# EPICS SNL sequencer program: mpgSupport/src/edefMask.st
program edefMask

option -a;  /* All pvGets must be synchronous */
option +c;  /* All connections must be made before execution begins */
option +d;  /* Turn on runtime debug messages */

%%#include <string.h> 	   /* sprintf prototype */

int maskChanged;
assign maskChanged to "{IOC}:MASKCHG";
monitor maskChanged;
evflag maskChanged_ef;
sync maskChanged maskChanged_ef;

int bitChanged;
assign bitChanged to "{IOC}:BITCHG";
monitor bitChanged;
evflag bitChanged_ef;
sync bitChanged bitChanged_ef;

unsigned long dgrpINCM[3];
assign dgrpINCM to "VX00:DGRP:1150:INCM";
monitor dgrpINCM;

unsigned long dgrpEXCM[3];
assign dgrpEXCM to "VX00:DGRP:1150:EXCM";
monitor dgrpEXCM;

int initDone;
assign initDone to "{IOC}:MASKSETUP";

unsigned short dgrpSHORT;
short i;
short j;
short eachBit;
short bitp;
short savedINCM[20][160];
short savedEXCM[20][160];

int edefMaxNumber;
int edefNumber;

int maskMaxNumber;
int maskCount;
int maskNumber;
int maskVal;

int pnbnMaxNumber;
int pnbnNumber;

string NAMEval;
assign NAMEval to "";
string NAMEpv;

string PNBNval;
assign PNBNval to "";
string PNBNpv;

int BITPval;
assign BITPval to "";
string BITPpv;

int BITWval;
assign BITWval to "";
string BITWpv;

string DESCval;
assign DESCval to "";
string DESCpv;

string DESC1val;
assign DESC1val to "";
string DESC1pv;

int INCMval;
assign INCMval to "";
string INCMpv;

int EXCMval;
assign EXCMval to "";
string EXCMpv;

string INCMSval;
assign INCMSval to "";
string INCMSpv;
int iINCMS;

string EXCMSval;
assign EXCMSval to "";
string EXCMSpv;
int iEXCMS;

unsigned long INCLUSIONval;
assign INCLUSIONval to "";
string INCLUSIONpv;

unsigned long EXCLUSIONval;
assign EXCLUSIONval to "";
string EXCLUSIONpv;

unsigned short INCLUSIONvalSHORT;
assign INCLUSIONvalSHORT to "";
string INCLUSIONpvSHORT;

unsigned short EXCLUSIONvalSHORT;
assign EXCLUSIONvalSHORT to "";
string EXCLUSIONpvSHORT;

int sort_done;
int debug_flag;

char * SYS;

entry {

  debug_flag = 0;
  if (debug_flag) printf ("edefMask:entry\n");

  sort_done = 0;

  edefMaxNumber = 20;
  edefNumber = 0;

  maskMaxNumber = 160;
  maskCount = 0;
  maskNumber = 0;

  pnbnMaxNumber = 124;
  pnbnNumber = 0;
  sprintf (PNBNval, "");

  SYS = macValueGet("SYS");

  } /* edefMask entry*/

ss edefMaskStateSet {

  state pnbn_read {

    entry {
      if (debug_flag) printf ("edefMaskStateSet:pnbn_read");

      /* setup first PNBN NAME, BITP & BITW */
      pnbnNumber++;
      sprintf (PNBNpv, "MP00:PNBN:%d:NAME", pnbnNumber);
      pvAssign (PNBNval, PNBNpv);
      pvMonitor (PNBNval);

      BITPval = -1;
      sprintf (BITPpv, "MP00:PNBN:%d:BITP", pnbnNumber);
      pvAssign (BITPval, BITPpv);
      pvMonitor (BITPval);

      BITWval = -1;
      sprintf (BITWpv, "MP00:PNBN:%d:BITW", pnbnNumber);
      pvAssign (BITWval, BITWpv);
      pvMonitor (BITWval);
      } /* pnbn_read entry */

    when (pnbnNumber > pnbnMaxNumber) {
      } state pnbn_sort

    when ((strlen(PNBNval)>0) && (BITPval>-1) && (BITWval>-1)) {
      if ((BITPval < 32) || (0 == strncmp ("            ", PNBNval, 12))) {
        /* unused PNBN name, 32 comes from PNET_MODFBIT_LOLIM */
        }
      else {
        if (debug_flag) printf (".");
        maskCount++;
        /* Put the name in INCM DESC */
        sprintf (DESC1pv, "EDEF:%s:1:INCM%d.DESC", SYS, maskCount);
        pvAssign (DESC1val, DESC1pv);
        sprintf (DESC1val, "%s", PNBNval);
        pvPut (DESC1val);
        /* Put the BITP & BITW into the EXCM DESC */
        sprintf (DESC1pv, "EDEF:%s:1:EXCM%d.DESC", SYS, maskCount);
        pvAssign (DESC1val, DESC1pv);
        sprintf (DESC1val, "%3.3d %3.3d", BITPval, BITWval);
        pvPut (DESC1val);
        }; /* non-blank pnbn name */
      pnbnNumber++;
      sprintf (PNBNval, "");
      BITPval = -1;
      BITWval = -1;
      if (pnbnNumber <= pnbnMaxNumber) {
        sprintf (PNBNpv, "MP00:PNBN:%d:NAME", pnbnNumber);
        pvAssign (PNBNval, PNBNpv);
        pvMonitor (PNBNval);
        sprintf (BITPpv, "MP00:PNBN:%d:BITP", pnbnNumber);
        pvAssign (BITPval, BITPpv);
        pvMonitor (BITPval);
        sprintf (BITWpv, "MP00:PNBN:%d:BITW", pnbnNumber);
        pvAssign (BITWval, BITWpv);
        pvMonitor (BITWval);
        }; /* setup next pnbn unit */
      } state pnbn_read
    } /* state pnbn_read */

  state pnbn_sort {
    entry {
      if (debug_flag) printf ("\nedefMaskStateSet:pnbn_sort");
      }
    when (sort_done) {
      } state pnbn_assign
    when (1) {
      if (debug_flag) printf (".");
      sort_done = 1;
      for (maskNumber = 1; maskNumber < maskCount; maskNumber++) {
        sprintf (DESC1pv, "EDEF:%s:1:INCM%d.DESC", SYS, maskNumber);
        pvAssign (DESC1val, DESC1pv);
        pvGet (DESC1val);
        sprintf (DESCpv, "EDEF:%s:1:INCM%d.DESC", SYS, 1+maskNumber);
        pvAssign (DESCval, DESCpv);
        pvGet (DESCval);
        if (strcmp (DESC1val, DESCval) > 0) {
          sort_done = 0;
          /* switch INCM DESC's */
          sprintf (PNBNval, "%s", DESC1val);
          sprintf (DESC1val, "%s", DESCval);
          sprintf (DESCval, "%s", PNBNval);
          pvPut (DESC1val);
          pvPut (DESCval);
          /* switch EXCM DESC's */
          sprintf (DESC1pv, "EDEF:%s:1:EXCM%d.DESC", SYS, maskNumber);
          pvAssign (DESC1val, DESC1pv);
          pvGet (DESC1val);
          sprintf (DESCpv, "EDEF:%s:1:EXCM%d.DESC", SYS, 1+maskNumber);
          pvAssign (DESCval, DESCpv);
          pvGet (DESCval);
          sprintf (PNBNval, "%s", DESC1val);
          sprintf (DESC1val, "%s", DESCval);
          sprintf (DESCval, "%s", PNBNval);
          pvPut (DESC1val);
          pvPut (DESCval);
          }; /* switch */
        }; /* for each mask */
      } state pnbn_sort
    } /* state pnbn sort */

  state pnbn_assign {
    entry {
      if (debug_flag) printf ("\nedefMaskStateSet:pnbn_assign\n");
      }
    when (1) {
      for (maskNumber = 1; maskNumber <= maskCount; maskNumber++) {
        sprintf (DESC1pv, "EDEF:%s:1:INCM%d.DESC", SYS, maskNumber);
        pvAssign (DESC1val, DESC1pv);
        pvGet (DESC1val);
        for (edefNumber = 2; edefNumber <= edefMaxNumber; edefNumber++) {
          sprintf (DESCpv, "EDEF:%s:%d:INCM%d.DESC", SYS, edefNumber, maskNumber);
          pvAssign (DESCval, DESCpv);
          sprintf (DESCval, "%s", DESC1val);
          pvPut (DESCval);
          }; /* for each edef */
        }; /* for each mask */
      for (maskNumber = 1; maskNumber <= maskCount; maskNumber++) {
        sprintf (DESC1pv, "EDEF:%s:1:EXCM%d.DESC", SYS, maskNumber);
        pvAssign (DESC1val, DESC1pv);
        pvGet (DESC1val);
        for (edefNumber = 2; edefNumber <= edefMaxNumber; edefNumber++) {
          sprintf (DESCpv, "EDEF:%s:%d:EXCM%d.DESC", SYS, edefNumber, maskNumber);
          pvAssign (DESCval, DESCpv);
          sprintf (DESCval, "%s", DESC1val);
          pvPut (DESCval);
          }; /* for each edef */
        }; /* for each mask */
      } state dgrp_incm_excm_set
    } /* state pnbn assign */

  state dgrp_incm_excm_set {
    entry {
      if (debug_flag) printf ("edefMaskStateSet:dgrp_incm_excm_set\n");
      }
    /* read DGRP INCM & EXCM and set INCLUSION[1..5][A|B] & EXCLUSION[1..5][A|B] */
    when (1) {
      for (i=0; i<3; i++) {
        for (edefNumber = 1; edefNumber <= edefMaxNumber; edefNumber++) {
          dgrpSHORT = dgrpINCM[i] & 0x0000FFFF;
          sprintf (INCLUSIONpvSHORT, "EDEF:%s:%d:INCLUSION%dA", SYS, edefNumber, 1+i);
          pvAssign (INCLUSIONvalSHORT, INCLUSIONpvSHORT);
          INCLUSIONvalSHORT = dgrpSHORT;
          pvPut (INCLUSIONvalSHORT);

          dgrpSHORT = (dgrpINCM[i] & 0xFFFF0000) >> 16;
          sprintf (INCLUSIONpvSHORT, "EDEF:%s:%d:INCLUSION%dB", SYS, edefNumber, 1+i);
          pvAssign (INCLUSIONvalSHORT, INCLUSIONpvSHORT);
          INCLUSIONvalSHORT = dgrpSHORT;
          pvPut (INCLUSIONvalSHORT);

          dgrpSHORT = dgrpEXCM[i] & 0x0000FFFF;
          sprintf (EXCLUSIONpvSHORT, "EDEF:%s:%d:EXCLUSION%dA", SYS, edefNumber, 1+i);
          pvAssign (EXCLUSIONvalSHORT, EXCLUSIONpvSHORT);
          EXCLUSIONvalSHORT = dgrpSHORT;
          pvPut (EXCLUSIONvalSHORT);

          dgrpSHORT = (dgrpEXCM[i] & 0xFFFF0000) >> 16;
          sprintf (EXCLUSIONpvSHORT, "EDEF:%s:%d:EXCLUSION%dB", SYS, edefNumber, 1+i);
          pvAssign (EXCLUSIONvalSHORT, EXCLUSIONpvSHORT);
          EXCLUSIONvalSHORT = dgrpSHORT;
          pvPut (EXCLUSIONvalSHORT);
          }; /* for each edef */
        };
        sprintf (INCMSval, "1HZ");
        sprintf (PNBNval, "ONE_HERTZ");
      } state special_incm_excm_set
    } /* state dgrp_incm_excm_set */

  state special_incm_excm_set {
    /* Look for 1Hz and 10Hz eDefs and set their ONE_HERTZ & TEN_HERTZ INCLUSION[1..5][A|B] */
    entry {
      if (debug_flag) printf ("edefMaskStateSet:special_incm_excm_set\n");
      }
    when (0 == strlen(INCMSval)) {
      } state incm_excm_set
    when (1) {
      for (edefNumber = 1; edefNumber <= edefMaxNumber; edefNumber++) {
        sprintf (NAMEpv, "EDEF:%s:%d:NAME", SYS, edefNumber);
        pvAssign (NAMEval, NAMEpv);
        pvGet (NAMEval);
        if (0 == strncmp (NAMEval, INCMSval, strlen(INCMSval))) {
          for (maskNumber = 1; maskNumber <= maskCount; maskNumber++) {
            sprintf (DESCpv, "EDEF:%s:%d:INCM%d.DESC", SYS, edefNumber, maskNumber);
            pvAssign (DESCval, DESCpv);
            pvGet (DESCval);
            if (0 == strncmp (DESCval, PNBNval, strlen(PNBNval))) {
              sprintf (DESCpv, "EDEF:%s:%d:EXCM%d.DESC", SYS, edefNumber, maskNumber);
              pvAssign (DESCval, DESCpv);
              pvGet (DESCval);
              sscanf (DESCval, "%3d %3d", &BITPval, &BITWval);
              for (eachBit = 0; eachBit < BITWval; eachBit++) {
                bitp = BITPval + eachBit;
                j = 0; /* EDEF:SYS:[edefNumbner]:INCLUSION[j] */
                while (bitp > 31) {
                  j++;
                  bitp = bitp - 32;
                  };
                if (bitp < 16) {
                  sprintf (INCLUSIONpvSHORT, "EDEF:%s:%d:INCLUSION%dA", SYS, edefNumber, j);
                  pvAssign (INCLUSIONvalSHORT, INCLUSIONpvSHORT);
                  pvGet (INCLUSIONvalSHORT);
                  INCLUSIONvalSHORT += (1 << bitp);
                  pvPut (INCLUSIONvalSHORT);
                  }
                else {
                  sprintf (INCLUSIONpvSHORT, "EDEF:%s:%d:INCLUSION%dB", SYS, edefNumber, j);
                  pvAssign (INCLUSIONvalSHORT, INCLUSIONpvSHORT);
                  pvGet (INCLUSIONvalSHORT);
                  bitp = bitp - 16;
                  INCLUSIONvalSHORT += (1 << bitp);
                  pvPut (INCLUSIONvalSHORT);
                  };
                }; /* for each BITW */
              }; /* Found mask name */
            }; /* each mask */
          }; /* found correct EDEF NAME */
        }; /* each edef */
      if (0 == strcmp (INCMSval, "1HZ")) {
        sprintf (INCMSval, "10HZ");
        sprintf (PNBNval, "TEN_HERTZ");
        }
      else {
        sprintf (INCMSval, "");
        initDone = 1;
        pvPut (initDone);
        };
      } state special_incm_excm_set
    } /* state special_incm_excm */

  state incm_excm_set {
    /* Set INCMS[1..4] & EXCMS[1..4] and INCM[1..maskCount] & EXCM[1..maskCount]
       based on INCLUSION[1..5] EXCLUSION[1..5] */
    entry {
      if (debug_flag) printf ("edefMaskStateSet:incm_excm_set\n");
      }
    when(1) {
      for (edefNumber = 1; edefNumber <= edefMaxNumber; edefNumber++) {
        iINCMS=1;
        sprintf (INCMSpv, "EDEF:%s:%d:INCMS%d", SYS, edefNumber, iINCMS);
        pvAssign (INCMSval, INCMSpv);
        sprintf (INCMSval, "");
        iEXCMS=1;
        sprintf (EXCMSpv, "EDEF:%s:%d:EXCMS%d", SYS, edefNumber, iEXCMS);
        pvAssign (EXCMSval, EXCMSpv);
        sprintf (EXCMSval, "");
        for (maskNumber = 1; maskNumber <= maskCount; maskNumber++) {
          i = 0; /* index into INCLUSION & EXCLUSION */
          /* Is my BITP set? */
          sprintf (DESCpv, "EDEF:%s:%d:EXCM%d.DESC", SYS, edefNumber, maskNumber);
          pvAssign (DESCval, DESCpv);
          pvGet (DESCval);
          sscanf (DESCval, "%3d", &BITPval);
          sprintf (DESCpv, "EDEF:%s:%d:INCM%d.DESC", SYS, edefNumber, maskNumber);
          pvAssign (DESCval, DESCpv);
          pvGet (DESCval);
          sprintf (PNBNval, "%s", DESCval); /* remove trailing blanks */
          for (j=0; j<sizeof(PNBNval); j++) if (' ' == PNBNval[j]) PNBNval[j]=0;
          pvGet (DESCval);
          while (BITPval > 31) {
            i++;
            BITPval = BITPval - 32;
            };
          sprintf (INCLUSIONpv, "EDEF:%s:%d:INCLUSION%d", SYS, edefNumber, i);
          pvAssign (INCLUSIONval, INCLUSIONpv);
          pvGet (INCLUSIONval);
          sprintf (EXCLUSIONpv, "EDEF:%s:%d:EXCLUSION%d", SYS, edefNumber, i);
          pvAssign (EXCLUSIONval, EXCLUSIONpv);
          pvGet (EXCLUSIONval);
          sprintf (INCMpv, "EDEF:%s:%d:INCM%d", SYS, edefNumber, maskNumber);
          pvAssign (INCMval, INCMpv);
          pvGet (INCMval);
          sprintf (EXCMpv, "EDEF:%s:%d:EXCM%d", SYS, edefNumber, maskNumber);
          pvAssign (EXCMval, EXCMpv);
          pvGet (EXCMval);
          if (INCLUSIONval & (1 << BITPval)) {
            maskVal = 1;
            if ((strlen(INCMSval) + strlen(PNBNval)) > 38) {
              pvPut (INCMSval);
              sprintf (INCMSpv, "EDEF:%s:%d:INCMS%d", SYS, edefNumber, ++iINCMS);
              pvAssign (INCMSval, INCMSpv);
              sprintf (INCMSval, "");
              };
            if (iINCMS < 5) {
              if (0 == strlen(INCMSval)) {
                sprintf (INCMSval, "%s", PNBNval);
                }
              else {
                strcat (INCMSval, " ");
                strcat (INCMSval, PNBNval);
                };
              };
            } /* INCLUSION bit set */
          else {
            maskVal = 0;
            }; /* INCLUSION bit not set */
          if (maskVal != INCMval) {
            INCMval = maskVal;
            pvPut(INCMval);
            };
          if (EXCLUSIONval & (1 << BITPval)) {
            maskVal = 1;
            if ((strlen(EXCMSval) + strlen(PNBNval)) > 38) {
              pvPut (EXCMSval);
              sprintf (EXCMSpv, "EDEF:%s:%d:EXCMS%d", SYS, edefNumber, ++iEXCMS);
              pvAssign (EXCMSval, EXCMSpv);
              sprintf (EXCMSval, "");
              };
            if (iEXCMS < 5) {
              if (0 == strlen(EXCMSval)) {
                sprintf (EXCMSval, "%s", PNBNval);
                }
              else {
                strcat (EXCMSval, " ");
                strcat (EXCMSval, PNBNval);
                };
              };
            } /* EXCLUSION bit set */
          else {
            maskVal = 0;
            }; /* EXCLUSION bit not set */
          if (maskVal != EXCMval) {
            EXCMval = maskVal;
            pvPut(EXCMval);
            };
          }; /* for each Mask */
        while (iINCMS < 5) {
          pvPut (INCMSval);
          sprintf (INCMSpv, "EDEF:%s:%d:INCMS%d", SYS, edefNumber, ++iINCMS);
          pvAssign (INCMSval, INCMSpv);
          sprintf (INCMSval, "");
          };
        while (iEXCMS < 5) {
          pvPut (EXCMSval);
          sprintf (EXCMSpv, "EDEF:%s:%d:EXCMS%d", SYS, edefNumber, ++iEXCMS);
          pvAssign (EXCMSval, EXCMSpv);
          sprintf (EXCMSval, "");
          };
        }; /* for each edef */
      } state incm_excm_save
    } /* state incm_excm_set */

  state incm_excm_save {
    /* Save state of INCM[1..maskCount] & EXCM[1..maskCount] for later checking */
    entry {
      if (debug_flag) printf ("edefMaskStateSet:incm_excm_save\n");
      }
    when(1) {
      for (edefNumber = 1; edefNumber <= edefMaxNumber; edefNumber++) {
        for (maskNumber = 1; maskNumber <= maskCount; maskNumber++) {
          sprintf (INCMpv, "EDEF:%s:%d:INCM%d", SYS, edefNumber, maskNumber);
          pvAssign (INCMval, INCMpv);
          pvGet (INCMval);
          savedINCM[edefNumber-1][maskNumber-1] = INCMval;
          sprintf (EXCMpv, "EDEF:%s:%d:EXCM%d", SYS, edefNumber, maskNumber);
          pvAssign (EXCMval, EXCMpv);
          pvGet (EXCMval);
          savedEXCM[edefNumber-1][maskNumber-1] = EXCMval;
          }; /* each mask */
        }; /* each edef */
      efClear (maskChanged_ef);
      efClear (bitChanged_ef);
      } state checking
    } /* state incm_excm_save */

  state checking {
    /* Check for changes in INCM[1..maskCount] & EXCM[1..maskCount] and set
       INCLUSION[1..5][A|B] & EXCLUSION[1..5][A|B] */
    entry {
      if (debug_flag) printf ("edefMaskStateSet:checking\n");
      }
    when (efTest(maskChanged_ef)) {
      } state incm_excm_set
    when (efTest(bitChanged_ef)) {
      for (edefNumber = 1; edefNumber <= edefMaxNumber; edefNumber++) {
        for (maskNumber = 1; maskNumber <= maskCount; maskNumber++) {
          sprintf (INCMpv, "EDEF:%s:%d:INCM%d", SYS, edefNumber, maskNumber);
          pvAssign (INCMval, INCMpv);
          pvGet (INCMval);
          if (savedINCM[edefNumber-1][maskNumber-1] != INCMval) {
            /* Set INCLUSION[1..5][A|B] */
            sprintf (DESCpv, "EDEF:%s:%d:EXCM%d.DESC", SYS, edefNumber, maskNumber);
            pvAssign (DESCval, DESCpv);
            pvGet (DESCval);
            sscanf (DESCval, "%3d %3d", &BITPval, &BITWval);
            for (eachBit = 0; eachBit < BITWval; eachBit++) {
              bitp = BITPval + eachBit;
              j = 0; /* EDEF:SYS:[edefNumbner]:INCLUSION[j] */
              while (bitp > 31) {
                j++;
                bitp = bitp - 32;
                };
              if (bitp < 16) {
                sprintf (INCLUSIONpvSHORT, "EDEF:%s:%d:INCLUSION%dA", SYS, edefNumber, j);
                pvAssign (INCLUSIONvalSHORT, INCLUSIONpvSHORT);
                pvGet (INCLUSIONvalSHORT);
                if (INCMval) {
                  if (! (INCLUSIONvalSHORT & (1 << bitp))) INCLUSIONvalSHORT += (1 << bitp);
                  }
                else {
                  if (INCLUSIONvalSHORT & (1 << bitp)) INCLUSIONvalSHORT = INCLUSIONvalSHORT - (1 << bitp);
                  }
                pvPut (INCLUSIONvalSHORT);
                }
              else {
                sprintf (INCLUSIONpvSHORT, "EDEF:%s:%d:INCLUSION%dB", SYS, edefNumber, j);
                pvAssign (INCLUSIONvalSHORT, INCLUSIONpvSHORT);
                pvGet (INCLUSIONvalSHORT);
                bitp = bitp - 16;
                if (INCMval) {
                  if (! (INCLUSIONvalSHORT & (1 << bitp))) INCLUSIONvalSHORT += (1 << bitp);
                  }
                else {
                  if (INCLUSIONvalSHORT & (1 << bitp)) INCLUSIONvalSHORT = INCLUSIONvalSHORT - (1 << bitp);
                  };
                pvPut (INCLUSIONvalSHORT);
                };
              }; /* for each BITW */
            }; /* Set INCLUSION[1..5][A|B] */

          sprintf (EXCMpv, "EDEF:%s:%d:EXCM%d", SYS, edefNumber, maskNumber);
          pvAssign (EXCMval, EXCMpv);
          pvGet (EXCMval);
          if (savedEXCM[edefNumber-1][maskNumber-1] != EXCMval) {
            /* Set EXCLUSION[1..5][A|B] */
            sprintf (DESCpv, "EDEF:%s:%d:EXCM%d.DESC", SYS, edefNumber, maskNumber);
            pvAssign (DESCval, DESCpv);
            pvGet (DESCval);
            sscanf (DESCval, "%3d %3d", &BITPval, &BITWval);
            for (eachBit = 0; eachBit < BITWval; eachBit++) {
              bitp = BITPval + eachBit;
              j = 0; /* EDEF:SYS:[edefNumbner]:EXCLUSION[j] */
              while (bitp > 31) {
                j++;
                bitp = bitp - 32;
                };
              if (bitp < 16) {
                sprintf (EXCLUSIONpvSHORT, "EDEF:%s:%d:EXCLUSION%dA", SYS, edefNumber, j);
                pvAssign (EXCLUSIONvalSHORT, EXCLUSIONpvSHORT);
                pvGet (EXCLUSIONvalSHORT);
                if (EXCMval) {
                  if (! (EXCLUSIONvalSHORT & (1 << bitp))) EXCLUSIONvalSHORT += (1 << bitp);
                  }
                else {
                  if (EXCLUSIONvalSHORT & (1 << bitp)) EXCLUSIONvalSHORT = EXCLUSIONvalSHORT - (1 << bitp);
                  }
                pvPut (EXCLUSIONvalSHORT);
                }
              else {
                sprintf (EXCLUSIONpvSHORT, "EDEF:%s:%d:EXCLUSION%dB", SYS, edefNumber, j);
                pvAssign (EXCLUSIONvalSHORT, EXCLUSIONpvSHORT);
                pvGet (EXCLUSIONvalSHORT);
                bitp = bitp - 16;
                if (EXCMval) {
                  if (! (EXCLUSIONvalSHORT & (1 << bitp))) EXCLUSIONvalSHORT += (1 << bitp);
                  }
                else {
                  if (EXCLUSIONvalSHORT & (1 << bitp)) EXCLUSIONvalSHORT = EXCLUSIONvalSHORT - (1 << bitp);
                  };
                pvPut (EXCLUSIONvalSHORT);
                };
              }; /* for each BITW */
            }; /* Set EXCLUSION[1..5][A|B] */
          }; /* each mask */
        }; /* each edef */
      } state incm_excm_set
    } /* state checking */

} /* ss edefMaskStateSet */
